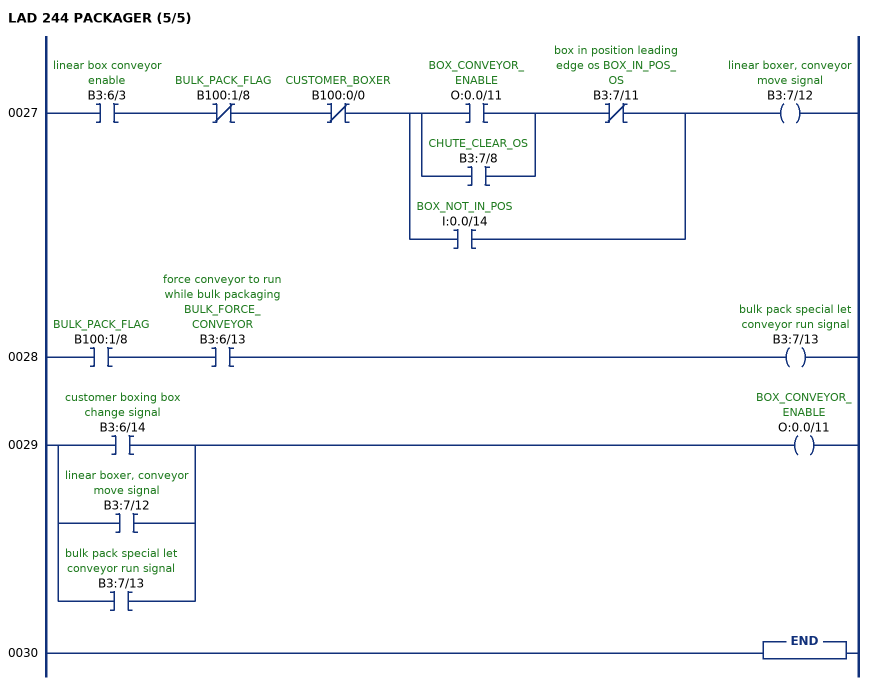
% Rung: 27 %
SOR XIC B3:6/3 XIO B100:1/8 XIO B100:0/0 BST BST XIC O:0.0/11 NXB XIC B3:7/8 BND XIO B3:7/11 NXB XIC I:0.0/14 BND OTE B3:7/12 EOR
%   B3:6/3  "linear box conveyor enable" %
%   B100:1/8  BULK_PACK_FLAG %
%   B100:0/0  CUSTOMER_BOXER %
%   O:0.0/11  BOX_CONVEYOR_ENABLE %
%   B3:7/8  CHUTE_CLEAR_OS %
%   B3:7/11  BOX_IN_POS_OS  "box in position leading edge os" %
%   I:0.0/14  BOX_NOT_IN_POS %
%   B3:7/12  "linear boxer, conveyor move signal" %
% Rung: 28 %
SOR XIC B100:1/8 XIC B3:6/13 OTE B3:7/13 EOR
%   B100:1/8  BULK_PACK_FLAG %
%   B3:6/13  BULK_FORCE_CONVEYOR  "force conveyor to run while bulk packaging" %
%   B3:7/13  "bulk pack special let conveyor run signal" %
% Rung: 29 %
SOR BST XIC B3:6/14 NXB XIC B3:7/12 NXB XIC B3:7/13 BND OTE O:0.0/11 EOR
%   B3:6/14  "customer boxing box change signal" %
%   B3:7/12  "linear boxer, conveyor move signal" %
%   B3:7/13  "bulk pack special let conveyor run signal" %
%   O:0.0/11  BOX_CONVEYOR_ENABLE %
% Rung: 30 %
SOR END EOR

LADDER 245 "NO PACKAGE"
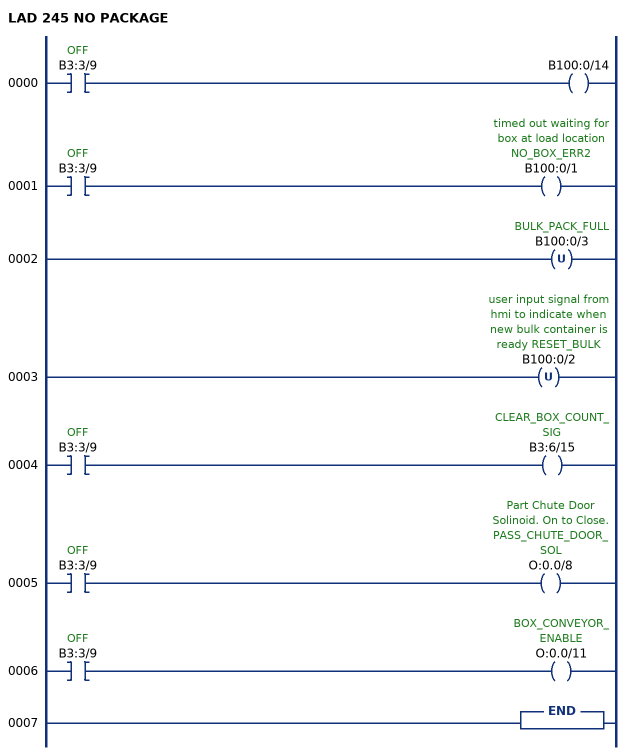
% Rung: 0 %
SOR XIC B3:3/9 OTE B100:0/14 EOR
%   B3:3/9  OFF %
% Rung: 1 %
SOR XIC B3:3/9 OTE B100:0/1 EOR
%   B3:3/9  OFF %
%   B100:0/1  NO_BOX_ERR2  "timed out waiting for box at load location" %
% Rung: 2 %
SOR OTU B100:0/3 EOR
%   B100:0/3  BULK_PACK_FULL %
% Rung: 3 %
SOR OTU B100:0/2 EOR
%   B100:0/2  RESET_BULK  "user input signal from hmi to indicate when new bulk container is ready" %
% Rung: 4 %
SOR XIC B3:3/9 OTE B3:6/15 EOR
%   B3:3/9  OFF %
%   B3:6/15  CLEAR_BOX_COUNT_SIG %
% Rung: 5 %
SOR XIC B3:3/9 OTE O:0.0/8 EOR
%   B3:3/9  OFF %
%   O:0.0/8  PASS_CHUTE_DOOR_SOL  "Part Chute Door Solinoid. On to Close." %
% Rung: 6 %
SOR XIC B3:3/9 OTE O:0.0/11 EOR
%   B3:3/9  OFF %
%   O:0.0/11  BOX_CONVEYOR_ENABLE %
% Rung: 7 %
SOR END EOR

LADDER 246 "RATE1"
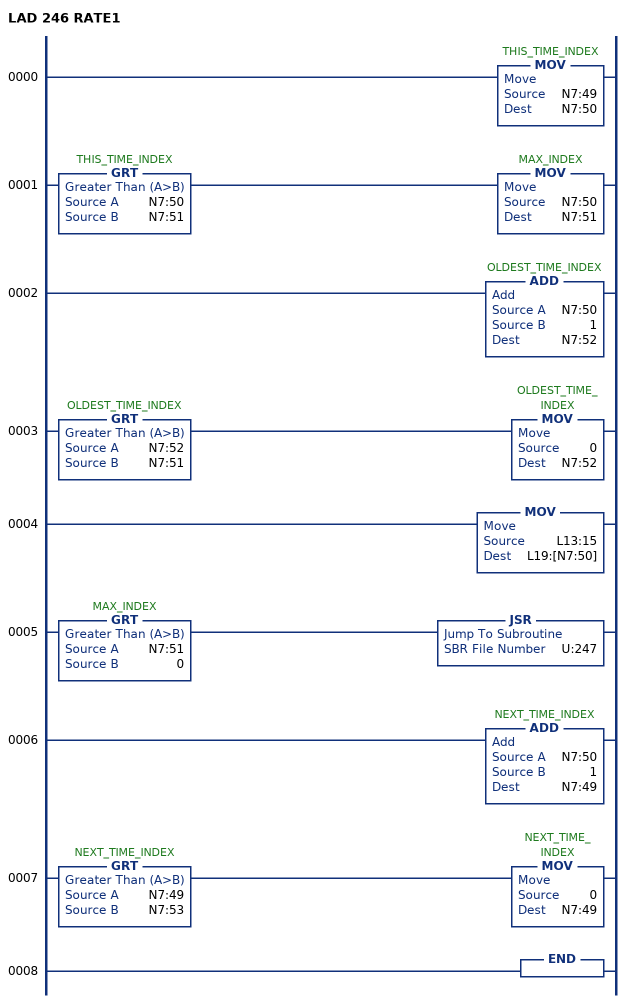
% Rung: 0 %
SOR MOV N7:49 N7:50 EOR
%   N7:49  NEXT_TIME_INDEX %
%   N7:50  THIS_TIME_INDEX %
% Rung: 1 %
SOR GRT N7:50 N7:51 MOV N7:50 N7:51 EOR
%   N7:50  THIS_TIME_INDEX %
%   N7:51  MAX_INDEX %
% Rung: 2 %
SOR ADD N7:50 1 N7:52 EOR
%   N7:50  THIS_TIME_INDEX %
%   N7:52  OLDEST_TIME_INDEX %
% Rung: 3 %
SOR GRT N7:52 N7:51 MOV 0 N7:52 EOR
%   N7:52  OLDEST_TIME_INDEX %
%   N7:51  MAX_INDEX %
% Rung: 4 %
SOR MOV L13:15 L19:[N7:50] EOR
%   L13:15  THE_TIME %
%   N7:50  THIS_TIME_INDEX %
% Rung: 5 %
SOR GRT N7:51 0 JSR U:247 EOR
%   N7:51  MAX_INDEX %
% Rung: 6 %
SOR ADD N7:50 1 N7:49 EOR
%   N7:50  THIS_TIME_INDEX %
%   N7:49  NEXT_TIME_INDEX %
% Rung: 7 %
SOR GRT N7:49 N7:53 MOV 0 N7:49 EOR
%   N7:49  NEXT_TIME_INDEX %
%   N7:53  UPPER_INDEX_LIMIT %
% Rung: 8 %
SOR END EOR

LADDER 247 "RATE2"
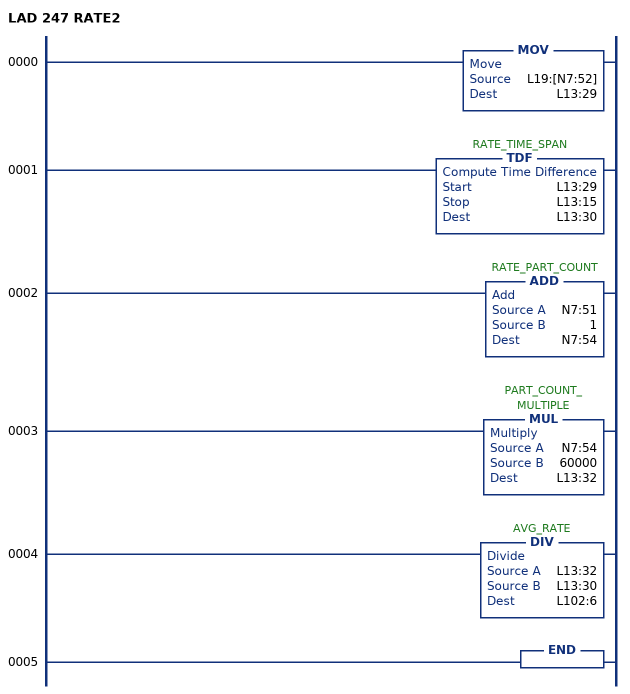
% Rung: 0 %
SOR MOV L19:[N7:52] L13:29 EOR
%   N7:52  OLDEST_TIME_INDEX %
% Rung: 1 %
SOR TDF L13:29 L13:15 L13:30 EOR
%   L13:15  THE_TIME %
%   L13:30  RATE_TIME_SPAN %
% Rung: 2 %
SOR ADD N7:51 1 N7:54 EOR
%   N7:51  MAX_INDEX %
%   N7:54  RATE_PART_COUNT %
% Rung: 3 %
SOR MUL N7:54 60000 L13:32 EOR
%   N7:54  RATE_PART_COUNT %
%   L13:32  PART_COUNT_MULTIPLE %
% Rung: 4 %
SOR DIV L13:32 L13:30 L102:6 EOR
%   L13:32  PART_COUNT_MULTIPLE %
%   L13:30  RATE_TIME_SPAN %
%   L102:6  AVG_RATE %
% Rung: 5 %
SOR END EOR

LADDER 248 "RESET RATE"
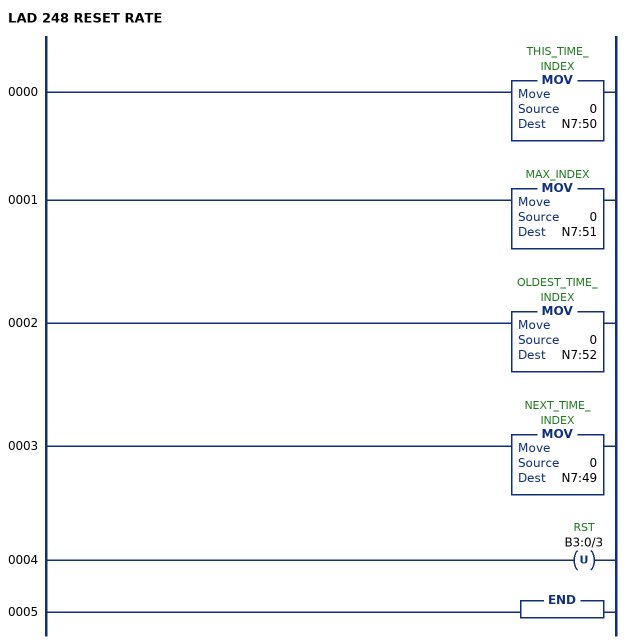
% Rung: 0 %
SOR MOV 0 N7:50 EOR
%   N7:50  THIS_TIME_INDEX %
% Rung: 1 %
SOR MOV 0 N7:51 EOR
%   N7:51  MAX_INDEX %
% Rung: 2 %
SOR MOV 0 N7:52 EOR
%   N7:52  OLDEST_TIME_INDEX %
% Rung: 3 %
SOR MOV 0 N7:49 EOR
%   N7:49  NEXT_TIME_INDEX %
% Rung: 4 %
SOR OTU B3:0/3 EOR
%   B3:0/3  RST %
% Rung: 5 %
SOR END EOR

LADDER 249 "NP STOP"    % stop on no good %
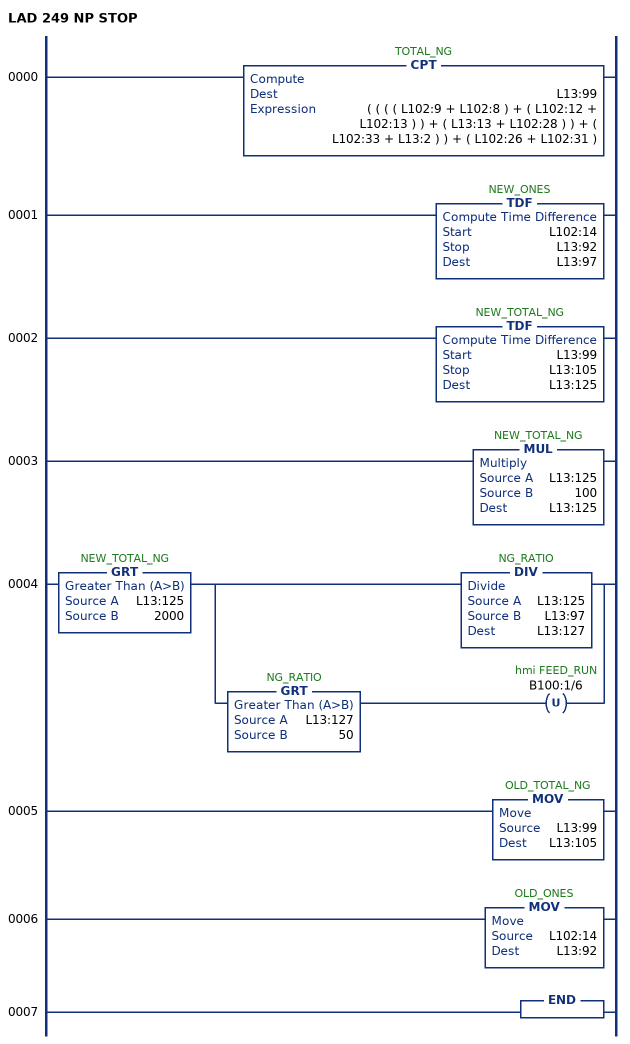
% Rung: 0 %
SOR CPT L13:99 " ( ( ( ( L102:9 + L102:8 ) + ( L102:12 + L102:13 ) ) + ( L13:13 + L102:28 ) ) + ( L102:33 + L13:2 ) ) + ( L102:26 + L102:31 ) " EOR
%   L13:99  TOTAL_NG %
%   L102:9  "too wide bottom" %
%   L102:8  "too close bottom" %
%   L102:12  "too close top count" %
%   L102:13  "too wide top count" %
%   L102:28  I1_I5_SKIPPEDCOUNT %
%   L102:33  I2_I6_SKIPPEDCOUNT %
%   L102:26  I1_I5_FAIL_COUNT %
%   L102:31  I2_I6_FAIL_COUNT %
% Rung: 1 %
SOR TDF L102:14 L13:92 L13:97 EOR
%   L102:14  ONES %
%   L13:92  OLD_ONES %
%   L13:97  NEW_ONES %
% Rung: 2 %
SOR TDF L13:99 L13:105 L13:125 EOR
%   L13:99  TOTAL_NG %
%   L13:105  OLD_TOTAL_NG %
%   L13:125  NEW_TOTAL_NG %
% Rung: 3 %
SOR MUL L13:125 100 L13:125 EOR
%   L13:125  NEW_TOTAL_NG %
% Rung: 4 %
SOR GRT L13:125 2000 BST DIV L13:125 L13:97 L13:127 NXB GRT L13:127 50 OTU B100:1/6 BND EOR
%   L13:125  NEW_TOTAL_NG %
%   L13:97  NEW_ONES %
%   L13:127  NG_RATIO %
%   B100:1/6  FEED_RUN  "hmi" %
% Rung: 5 %
SOR MOV L13:99 L13:105 EOR
%   L13:99  TOTAL_NG %
%   L13:105  OLD_TOTAL_NG %
% Rung: 6 %
SOR MOV L102:14 L13:92 EOR
%   L102:14  ONES %
%   L13:92  OLD_ONES %
% Rung: 7 %
SOR END EOR

LADDER 250 "SPEED BOT"    % high speed %
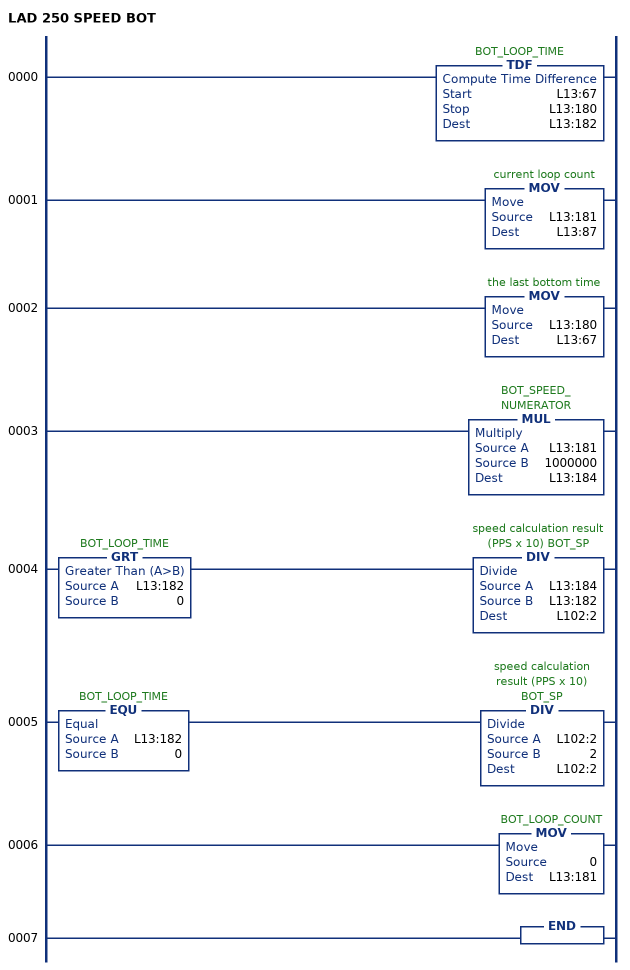
% Rung: 0 %
SOR TDF L13:67 L13:180 L13:182 EOR
%   L13:67  "the last bottom time" %
%   L13:180  BOT_THIS_TIME  "rtc bot belt movement event time" %
%   L13:182  BOT_LOOP_TIME %
% Rung: 1 %
SOR MOV L13:181 L13:87 EOR
%   L13:181  BOT_LOOP_COUNT %
%   L13:87  "current loop count" %
% Rung: 2 %
SOR MOV L13:180 L13:67 EOR
%   L13:180  BOT_THIS_TIME  "rtc bot belt movement event time" %
%   L13:67  "the last bottom time" %
% Rung: 3 %
SOR MUL L13:181 1000000 L13:184 EOR
%   L13:181  BOT_LOOP_COUNT %
%   L13:184  BOT_SPEED_NUMERATOR %
% Rung: 4 %
SOR GRT L13:182 0 DIV L13:184 L13:182 L102:2 EOR
%   L13:182  BOT_LOOP_TIME %
%   L13:184  BOT_SPEED_NUMERATOR %
%   L102:2  BOT_SP  "speed calculation result (PPS x 10)" %
% Rung: 5 %
SOR EQU L13:182 0 DIV L102:2 2 L102:2 EOR
%   L13:182  BOT_LOOP_TIME %
%   L102:2  BOT_SP  "speed calculation result (PPS x 10)" %
% Rung: 6 %
SOR MOV 0 L13:181 EOR
%   L13:181  BOT_LOOP_COUNT %
% Rung: 7 %
SOR END EOR

LADDER 251 "SPEED TOP"    % high speed %
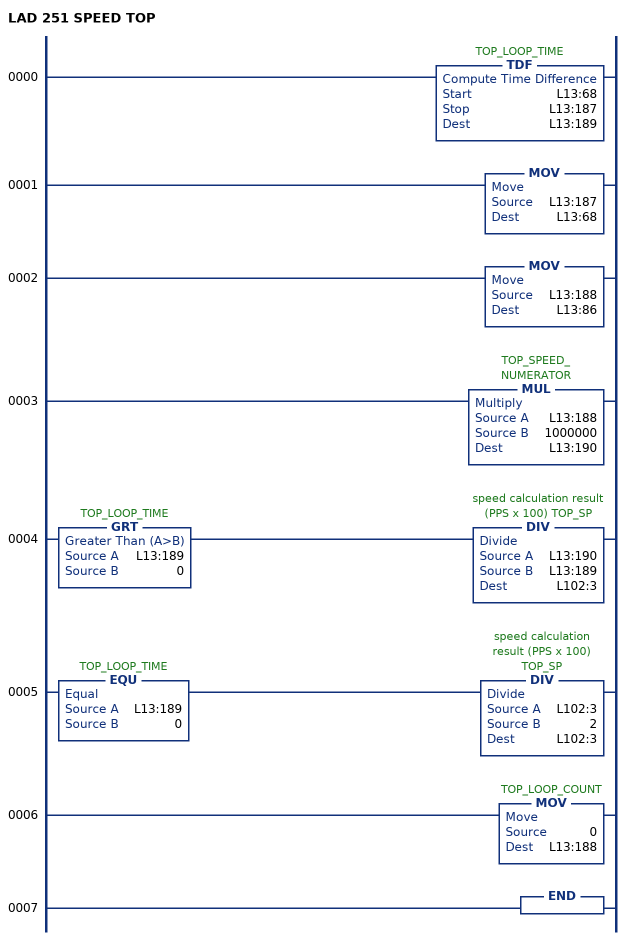
% Rung: 0 %
SOR TDF L13:68 L13:187 L13:189 EOR
%   L13:187  TOP_THIS_TIME  "rtc top belt movement event time" %
%   L13:189  TOP_LOOP_TIME %
% Rung: 1 %
SOR MOV L13:187 L13:68 EOR
%   L13:187  TOP_THIS_TIME  "rtc top belt movement event time" %
% Rung: 2 %
SOR MOV L13:188 L13:86 EOR
%   L13:188  TOP_LOOP_COUNT %
% Rung: 3 %
SOR MUL L13:188 1000000 L13:190 EOR
%   L13:188  TOP_LOOP_COUNT %
%   L13:190  TOP_SPEED_NUMERATOR %
% Rung: 4 %
SOR GRT L13:189 0 DIV L13:190 L13:189 L102:3 EOR
%   L13:189  TOP_LOOP_TIME %
%   L13:190  TOP_SPEED_NUMERATOR %
%   L102:3  TOP_SP  "speed calculation result (PPS x 100)" %
% Rung: 5 %
SOR EQU L13:189 0 DIV L102:3 2 L102:3 EOR
%   L13:189  TOP_LOOP_TIME %
%   L102:3  TOP_SP  "speed calculation result (PPS x 100)" %
% Rung: 6 %
SOR MOV 0 L13:188 EOR
%   L13:188  TOP_LOOP_COUNT %
% Rung: 7 %
SOR END EOR

LADDER 252 "P BOT"    % high speed %
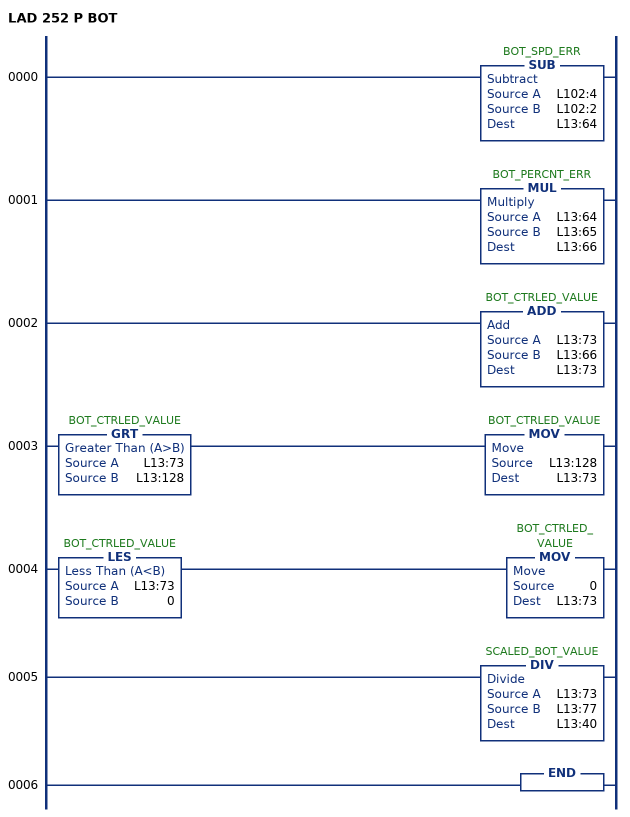
% Rung: 0 %
SOR SUB L102:4 L102:2 L13:64 EOR
%   L102:4  BOT_SPD_SETPOINT %
%   L102:2  BOT_SP  "speed calculation result (PPS x 10)" %
%   L13:64  BOT_SPD_ERR %
% Rung: 1 %
SOR MUL L13:64 L13:65 L13:66 EOR
%   L13:64  BOT_SPD_ERR %
%   L13:65  POS5SHIFT %
%   L13:66  BOT_PERCNT_ERR %
% Rung: 2 %
SOR ADD L13:73 L13:66 L13:73 EOR
%   L13:73  BOT_CTRLED_VALUE %
%   L13:66  BOT_PERCNT_ERR %
% Rung: 3 %
SOR GRT L13:73 L13:128 MOV L13:128 L13:73 EOR
%   L13:73  BOT_CTRLED_VALUE %
%   L13:128  "how much top has shifted since measurment" %
% Rung: 4 %
SOR LES L13:73 0 MOV 0 L13:73 EOR
%   L13:73  BOT_CTRLED_VALUE %
% Rung: 5 %
SOR DIV L13:73 L13:77 L13:40 EOR
%   L13:73  BOT_CTRLED_VALUE %
%   L13:40  SCALED_BOT_VALUE %
% Rung: 6 %
SOR END EOR

LADDER 253 "P TOP"    % high speed %
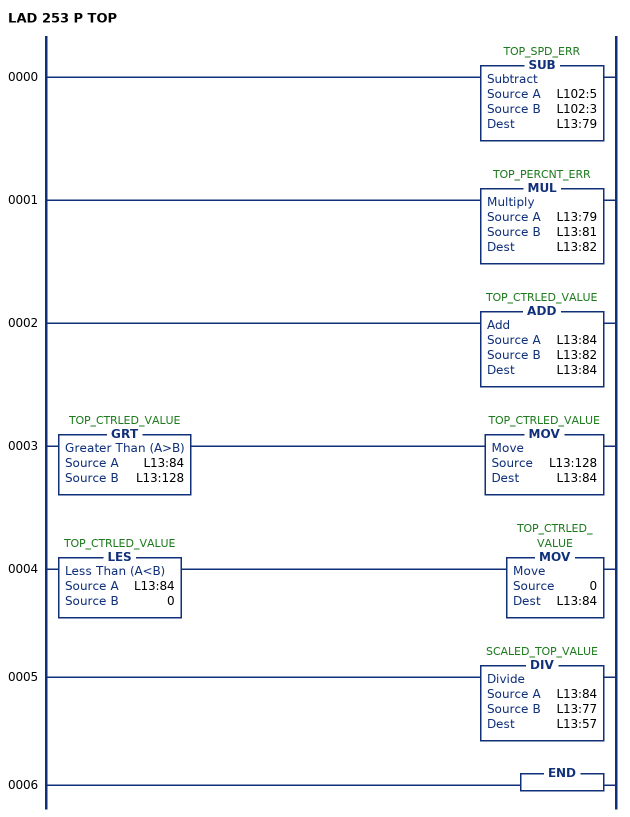
% Rung: 0 %
SOR SUB L102:5 L102:3 L13:79 EOR
%   L102:5  TOP_SPD_SETPOINT %
%   L102:3  TOP_SP  "speed calculation result (PPS x 100)" %
%   L13:79  TOP_SPD_ERR %
% Rung: 1 %
SOR MUL L13:79 L13:81 L13:82 EOR
%   L13:79  TOP_SPD_ERR %
%   L13:81  TOP_FDBK_RATIO %
%   L13:82  TOP_PERCNT_ERR %
% Rung: 2 %
SOR ADD L13:84 L13:82 L13:84 EOR
%   L13:84  TOP_CTRLED_VALUE %
%   L13:82  TOP_PERCNT_ERR %
% Rung: 3 %
SOR GRT L13:84 L13:128 MOV L13:128 L13:84 EOR
%   L13:84  TOP_CTRLED_VALUE %
%   L13:128  "how much top has shifted since measurment" %
% Rung: 4 %
SOR LES L13:84 0 MOV 0 L13:84 EOR
%   L13:84  TOP_CTRLED_VALUE %
% Rung: 5 %
SOR DIV L13:84 L13:77 L13:57 EOR
%   L13:84  TOP_CTRLED_VALUE %
%   L13:57  SCALED_TOP_VALUE %
% Rung: 6 %
SOR END EOR

LADDER 254 "TOTALCOUNT"
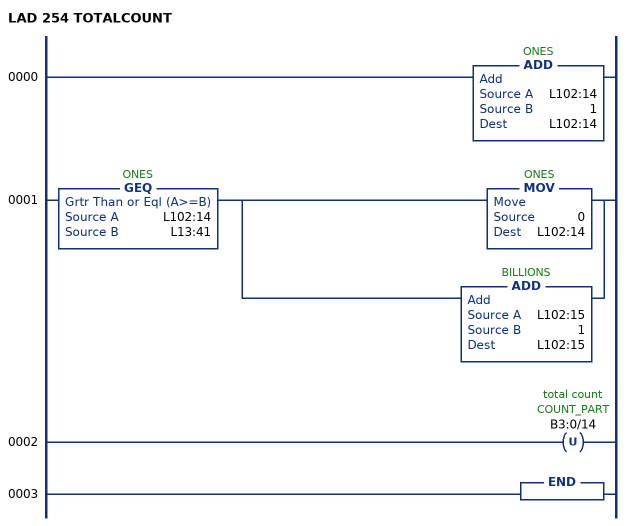
% Rung: 0 %
SOR ADD L102:14 1 L102:14 EOR
%   L102:14  ONES %
% Rung: 1 %
SOR GEQ L102:14 L13:41 BST MOV 0 L102:14 NXB ADD L102:15 1 L102:15 BND EOR
%   L102:14  ONES %
%   L13:41  "skipped count change in the last 3 seconds" %
%   L102:15  BILLIONS %
% Rung: 2 %
SOR OTU B3:0/14 EOR
%   B3:0/14  COUNT_PART  "total count" %
% Rung: 3 %
SOR END EOR

LADDER 255 "SAVED"
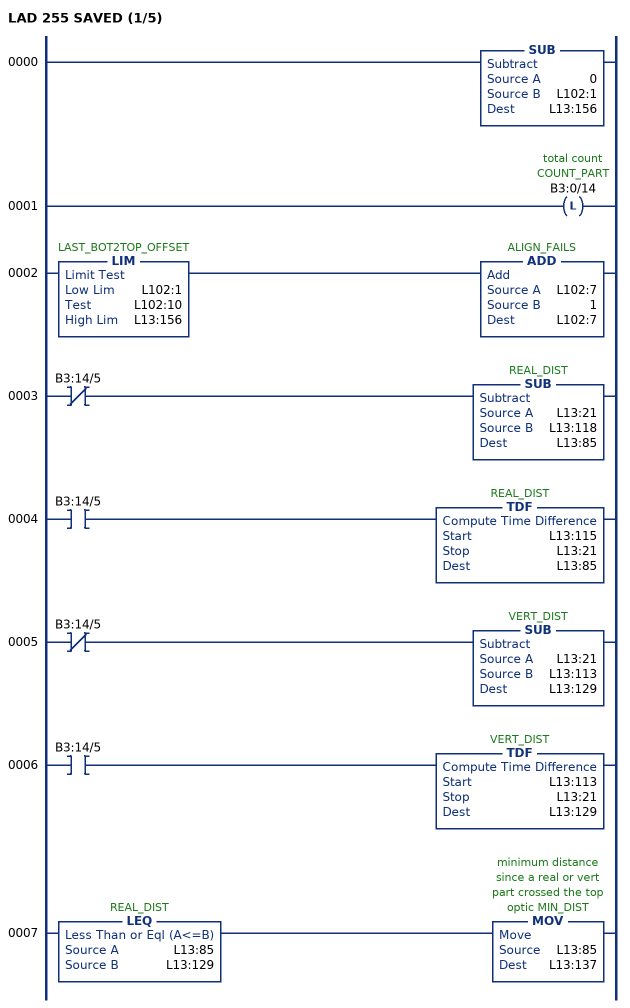
% Rung: 0 %
SOR SUB 0 L102:1 L13:156 EOR
%   L102:1  MAX_OFFSET  "transition zone width" %
% Rung: 1 %
SOR OTL B3:0/14 EOR
%   B3:0/14  COUNT_PART  "total count" %
% Rung: 2 %
SOR LIM L102:1 L102:10 L13:156 ADD L102:7 1 L102:7 EOR
%   L102:1  MAX_OFFSET  "transition zone width" %
%   L102:10  LAST_BOT2TOP_OFFSET %
%   L102:7  ALIGN_FAILS %
% Rung: 3 %
SOR XIO B3:14/5 SUB L13:21 L13:118 L13:85 EOR
%   L13:21  TOP_POSITION %
%   L13:118  REAL_CL_POSITION  "real part center line in raw position" %
%   L13:85  REAL_DIST %
% Rung: 4 %
SOR XIC B3:14/5 TDF L13:115 L13:21 L13:85 EOR
%   L13:115  TRAILING_EDGE_POS  "top optic trailing edge position" %
%   L13:21  TOP_POSITION %
%   L13:85  REAL_DIST %
% Rung: 5 %
SOR XIO B3:14/5 SUB L13:21 L13:113 L13:129 EOR
%   L13:21  TOP_POSITION %
%   L13:113  VIRT_CL_POSITION  "virtual part center line transfer from the bottom in raw position" %
%   L13:129  VERT_DIST %
% Rung: 6 %
SOR XIC B3:14/5 TDF L13:113 L13:21 L13:129 EOR
%   L13:113  VIRT_CL_POSITION  "virtual part center line transfer from the bottom in raw position" %
%   L13:21  TOP_POSITION %
%   L13:129  VERT_DIST %
% Rung: 7 %
SOR LEQ L13:85 L13:129 MOV L13:85 L13:137 EOR
%   L13:85  REAL_DIST %
%   L13:129  VERT_DIST %
%   L13:137  MIN_DIST  "minimum distance since a real or vert part crossed the top optic" %

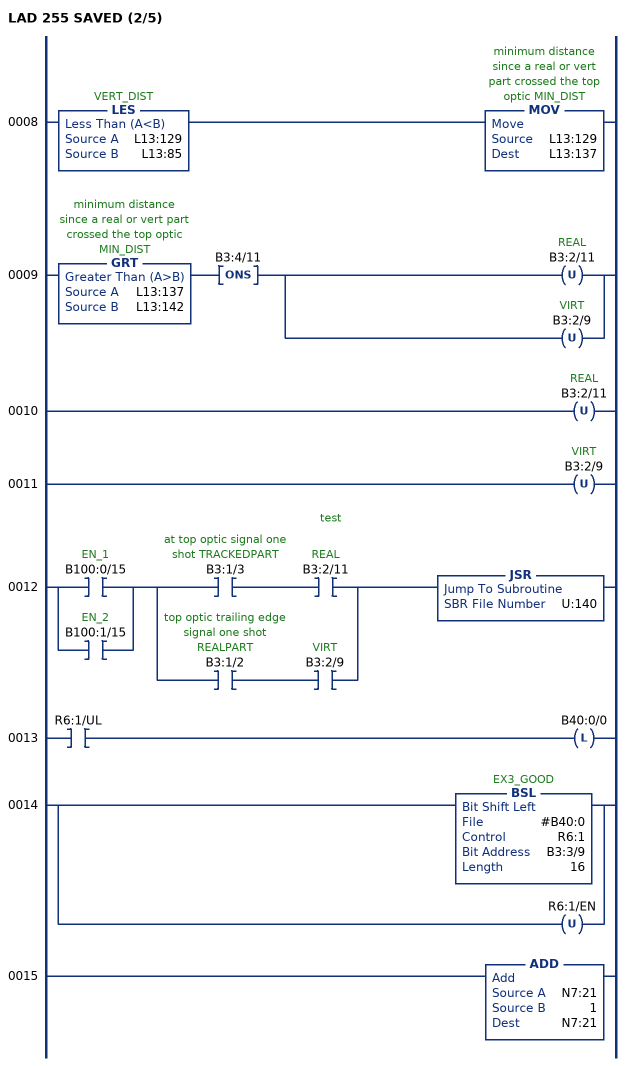
% Rung: 8 %
SOR LES L13:129 L13:85 MOV L13:129 L13:137 EOR
%   L13:129  VERT_DIST %
%   L13:85  REAL_DIST %
%   L13:137  MIN_DIST  "minimum distance since a real or vert part crossed the top optic" %
% Rung: 9 %
SOR GRT L13:137 L13:142 ONS B3:4/11 BST OTU B3:2/11 NXB OTU B3:2/9 BND EOR
%   L13:137  MIN_DIST  "minimum distance since a real or vert part crossed the top optic" %
%   L13:142  LAST_ALIGNMENT_FAILS %
%   B3:2/11  REAL %
%   B3:2/9  VIRT %
% Rung: 10 %
SOR OTU B3:2/11 EOR
%   B3:2/11  REAL %
% Rung: 11 %
SOR OTU B3:2/9 EOR
%   B3:2/9  VIRT %
% Rung: 12 %
% test %
SOR BST XIC B100:0/15 NXB XIC B100:1/15 BND BST XIC B3:1/3 XIC B3:2/11 NXB XIC B3:1/2 XIC B3:2/9 BND JSR U:140 EOR
%   B100:0/15  EN_1 %
%   B100:1/15  EN_2 %
%   B3:1/3  TRACKEDPART  "at top optic signal one shot" %
%   B3:2/11  REAL %
%   B3:1/2  REALPART  "top optic trailing edge signal one shot" %
%   B3:2/9  VIRT %
% Rung: 13 %
SOR XIC R6:1/UL OTL B40:0/0 EOR
% Rung: 14 %
SOR BST BSL #B40:0 R6:1 B3:3/9 16 NXB OTU R6:1/EN BND EOR
%   B40:0  EX3_GOOD %
%   B3:3/9  OFF %
% Rung: 15 %
SOR ADD N7:21 1 N7:21 EOR

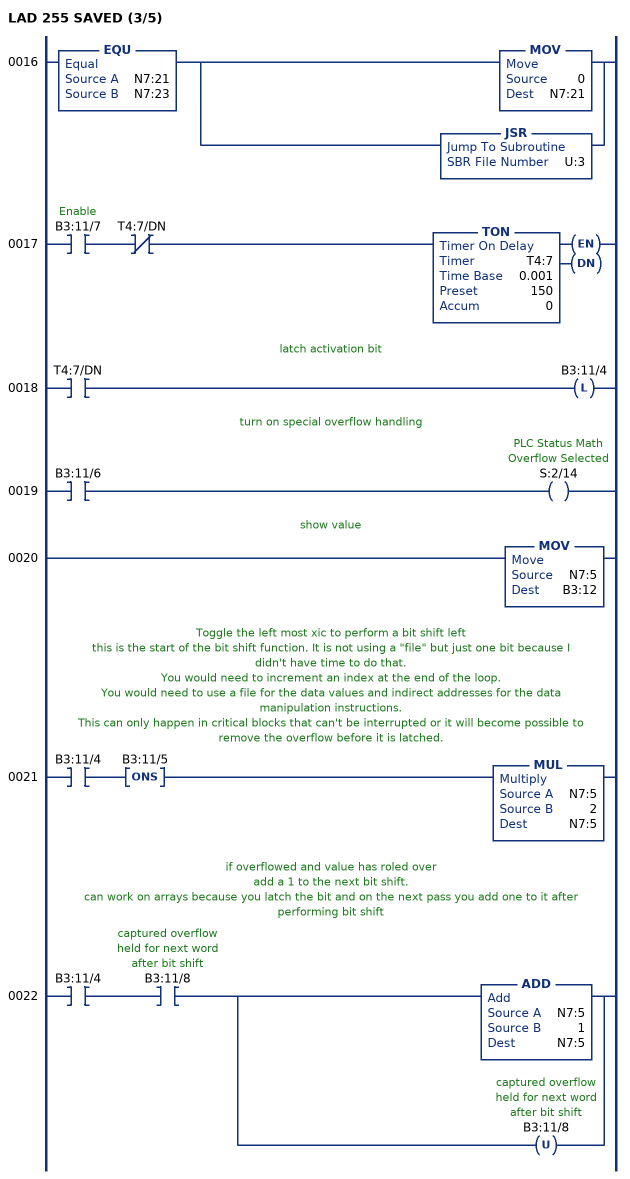
% Rung: 16 %
SOR EQU N7:21 N7:23 BST MOV 0 N7:21 NXB JSR U:3 BND EOR
% Rung: 17 %
SOR XIC B3:11/7 XIO T4:7/DN TON T4:7 0.001 150 0 EOR
%   B3:11/7  "Enable" %
% Rung: 18 %
% latch activation bit %
SOR XIC T4:7/DN OTL B3:11/4 EOR
% Rung: 19 %
% turn on special overflow handling %
SOR XIC B3:11/6 OTE S:2/14 EOR
%   S:2/14  "PLC Status Math Overflow Selected" %
% Rung: 20 %
% show value %
SOR MOV N7:5 B3:12 EOR
% Rung: 21 %
% Toggle the left most xic to perform a bit shift left
% 
% this is the start of the bit shift function. It is not using a "file" but just one bit because I didn't have time to do that.
% You would need to increment an index at the end of the loop.
% You would need to use a file for the data values and indirect addresses for the data manipulation instructions.
% 
% This can only happen in critical blocks that can't be interrupted or it will become possible to remove the overflow before it is latched. %
SOR XIC B3:11/4 ONS B3:11/5 MUL N7:5 2 N7:5 EOR
% Rung: 22 %
% if overflowed and value has roled over
% add a 1 to the next bit shift.
% can work on arrays because you latch the bit and on the next pass you add one to it after performing bit shift %
SOR XIC B3:11/4 XIC B3:11/8 BST ADD N7:5 1 N7:5 NXB OTU B3:11/8 BND EOR
%   B3:11/8  "captured overflow held for next word after bit shift" %

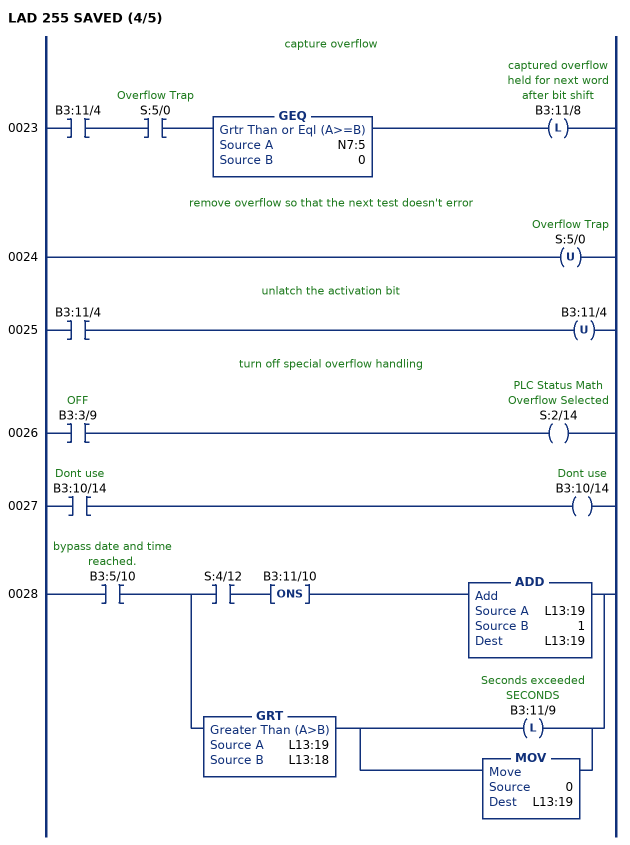
% Rung: 23 %
% capture overflow %
SOR XIC B3:11/4 XIC S:5/0 GEQ N7:5 0 OTL B3:11/8 EOR
%   S:5/0  "Overflow Trap" %
%   B3:11/8  "captured overflow held for next word after bit shift" %
% Rung: 24 %
% remove overflow so that the next test doesn't error %
SOR OTU S:5/0 EOR
%   S:5/0  "Overflow Trap" %
% Rung: 25 %
% unlatch the activation bit %
SOR XIC B3:11/4 OTU B3:11/4 EOR
% Rung: 26 %
% turn off special overflow handling %
SOR XIC B3:3/9 OTE S:2/14 EOR
%   B3:3/9  OFF %
%   S:2/14  "PLC Status Math Overflow Selected" %
% Rung: 27 %
SOR XIC B3:10/14 OTE B3:10/14 EOR
%   B3:10/14  "Dont use" %
% Rung: 28 %
SOR XIC B3:5/10 BST XIC S:4/12 ONS B3:11/10 ADD L13:19 1 L13:19 NXB GRT L13:19 L13:18 BST OTL B3:11/9 NXB MOV 0 L13:19 BND BND EOR
%   B3:5/10  "bypass date and time reached." %
%   L13:18  MAX %
%   B3:11/9  SECONDS  "Seconds exceeded" %

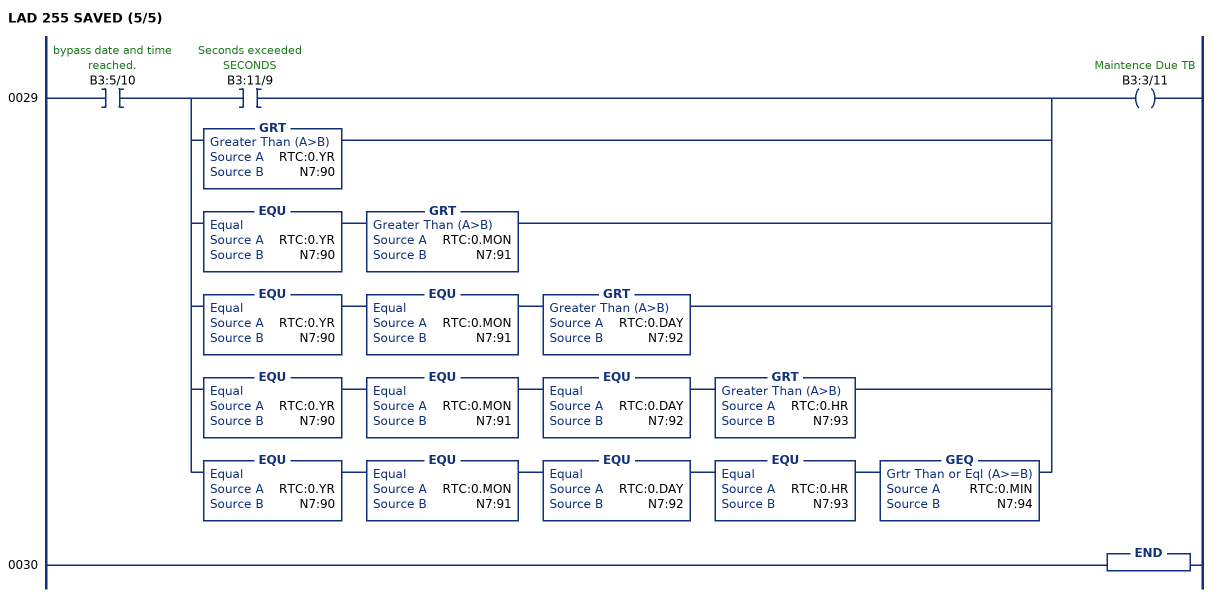
% Rung: 29 %
SOR XIC B3:5/10 BST XIC B3:11/9 NXB GRT RTC:0.YR N7:90 NXB EQU RTC:0.YR N7:90 GRT RTC:0.MON N7:91 NXB EQU RTC:0.YR N7:90 EQU RTC:0.MON N7:91 GRT RTC:0.DAY N7:92 NXB EQU RTC:0.YR N7:90 EQU RTC:0.MON N7:91 EQU RTC:0.DAY N7:92 GRT RTC:0.HR N7:93 NXB EQU RTC:0.YR N7:90 EQU RTC:0.MON N7:91 EQU RTC:0.DAY N7:92 EQU RTC:0.HR N7:93 GEQ RTC:0.MIN N7:94 BND OTE B3:3/11 EOR
%   B3:5/10  "bypass date and time reached." %
%   B3:11/9  SECONDS  "Seconds exceeded" %
%   N7:90  RTC %
%   B3:3/11  TB  "Maintence Due" %
% Rung: 30 %
SOR END EOR

OTHER DOCUMENTED ADDRESSES
  B38:0  EX1_GOOD
  B189:0/0  "change box"
  B189:0/9  "override boxing ok or not full signal"
  B189:0/11  "HMI force door close"
  B196:1/0  "Chute door is closed"
  B196:1/1  "control chute door"
  B196:1/13  "force box conveyor on"
  B196:3/0  "for hmi to continue production unlatched by hmi"
  HSC:0.0  "top"
  HSC:0.3/6  "Underflow interrupt"
  HSC:0.3/7  "Overflow interrupt"
  HSC:1.0  "bot"
  HSC:1.3/6  "Underflow interrupt"
  HSC:1.3/7  "Overflow interrupt"
  I7_TRAC  
  I:0.0/0  TOP_EN  "Encoder Signal Top"
  I:0.0/4  BOT_EN  "Encoder Signal Bot"
  I:0.1/4  "not used"
  I:0.1/5  "not used"
  I:0.1/6  "not used"
  I:0.1/7  "not used"
  I:0.1/8  "not used"
  I:0.1/9  "not used"
  I:0.1/10  "not used"
  I:0.1/11  "not used"
  I:0.1/12  "not used"
  I:0.1/13  "not used"
  I:0.1/14  "not used"
  I:0.1/15  "not used"
  I:0.2  "not used"
  I:0.3  "not used"
  I:0.4  "Spare Analog Input 1"
  I:0.5  "Spare Analog Input 2"
  I:0.6  "Spare Analog Input 3"
  I:2.0/0  FRONT_ESTOP
  I:2.0/1  REAR_ESTOP
  I:2.0/3  BOX_CNV_NOT_FULL  "input turns off when box discharge full optics are blocked"
  I:2.0/4  "this input is on when a box is not in position"
  I:2.0/8  FRONT_DOOR  "front door signal ce models only"
  I:2.0/9  REAR_DOOR  "rear door signal ce models only"
  I:2.0/11  "spare"
  L13:132  "set speed"
  L13:133  "controlled speed"
  L13:183  TKS_PER_SECOND
  L23:19  TOP_OPT_FAIL_CT
  L23:34  AIR_PRESSURE_FAULT
  L28:0  INS_1_TIME
  L29:0  INS_1_POS
  L30:0  INS_5_TIME
  L31:0  INS_5_POS
  L32:0  INS_6_TIME
  L33:0  INS_6_POS
  L192:1  BOT_LAST_TIME  "rtc bot belt previous movement event time"
  L192:2  BOT_CYCLE_TIME  "rtc bot belt time between events"
  L192:7  FROM_REAL  "distance from real part signal at optic location"
  L192:8  FROM_TRACKED  "distance from tracked part signal at optic location"
  L192:16  TOP_LAST_TIME  "rtc top belt previous movement event time"
  L192:17  TOP_CYCLE_TIME  "rtc top belt time between events"
  L199:5  ACQTM51
  L199:6  ACQTM52
  L199:7  ACQTM53
  L199:9  "ones"
  L199:10  "billions"
  L199:13  DUMP_LONG
  L199:15  ACQTM11
  L199:16  ACQTM12
  L199:17  ACQTM13
  L199:20  RESULTTM1
  L199:22  CLEARTIME5COUNT
  L199:23  CLEARTIME6COUNT
  L199:24  ACQTM61
  L199:25  ACQTM62
  L199:26  ACQTM63
  L199:27  TMSINCETRIG1
  L199:29  TMSINCETRIG5
  L199:30  TMSINCETRIG6
  L199:31  CLEARTIME1COUNT
  L199:32  RESULTTM5
  L199:33  RESULTTM6
  L199:34  MAXACQTM1
  L199:36  MAXACQTM6
  N7  
  N101:2  I3_TRIG_LOC
  N101:3  I4_TRIG_LOC
  O:0.0/1  "spare"
  O:0.0/12  "not used"
  O:0.0/13  "not used"
  O:0.0/14  "not used"
  O:0.0/15  "not used"
  O:0.1  "not used"
  O:0.2  "not used"
  O:0.3  "not used"
  O:1.2  "Feeder Bowl Speed"
  O:3.0/1  "Part Chute Door Solinoid. On to Close."
  O:3.0/2  "spare"
  O:3.0/3  "light curtain range selection /* needed? */"
  O:3.0/7  "door unlocks on CE models"
  O:3.0/8  "Light?"
  O:3.0/9  NUT_HOPPER  "Nut Hopper Enable"
  O:3.0/11  NUT_FEEDER_AIR  "Nut Feeder Bowl Air Enable"
  O:3.0/12  BOLT_FEEDER  "feeder bowl output on = enable"
  PFILE:6  "check for part jams"
  PFILE:10  "Bottom belt HSC"
  PFILE:12  "Top belt HSC"
  Q2:55  END_OF_MAIN
  Q5:94  END_OF_BELTS
  T20:0  "Trigger On Time"
  U:9  "slow data"
  U:24  "check skipped fail rate"
  U:28  "faults"
  U:29  "speed"
  U:30  "count"
  U:31  "rate calc"
  U:32  "boxer"
  U:33  "bulk pack"
  U:34  "customer boxing unit signals"
  U:35  "cleanup"

COMMENTS NOT ATTACHED TO A CURRENT RUNG
  R6:2: B41 is the top good 3 file
  R6:6/DN: B35 is the top NG file
  R6:10/DN: B37 is the top good 1 file
  R6:11/DN: B39 is the top good 2 file
  B100:1/15: what is this code for?
  R6:0: B36 is the bottom GOOD file
  R6:10: B37 is the top good 1 file
  R6:6: B35 is the top NG file
  R6:4: B34 is the bottom NG file

REVISION NOTES
  13: updated count reset
  14: added io moduals
  15: multiple steps toward new hmi integration
  21: test
  27: fix error if bulk pack and no boxing fallout were on

DATA TABLE (non-zero values as saved)
DATA B3
% B3:0 % 0X8862 0X1141 0X4041 0X6101 0XECB7 0X1504 0X0438 0X0461 0X3FA0 0X2330
% B3:10 % 0X21F0 0X40C6 0X4000 0X10B4 0X4801 0X0000 0X0000 0X0000 0X0000 0X0000
% B3:50 % 0X0001 0X0000 0X0000 0X0000 0X0000 0X0000 0X0000 0X0000 0X0000 0X0000
DATA T4
% .PRE .ACC %
% T4:0 % 0 1
% T4:1 % 150 0
% T4:2 % 400 0
% T4:3 % 250 68
% T4:4 % 1000 1000
% T4:5 % 5 5
% T4:6 % 10 32766
% T4:7 % 150 0
% T4:8 % 20 0
% T4:9 % 50 34
% T4:10 % 200 200
% T4:11 % 111 0
% T4:12 % 30 30
% T4:13 % 250 0
% T4:14 % 666 0
% T4:15 % 1000 1002
% T4:16 % 400 0
% T4:17 % 100 11
% T4:18 % 5 0
% T4:19 % 300 0
% T4:20 % 200 0
% T4:21 % 200 0
% T4:22 % 200 0
% T4:23 % 250 0
% T4:24 % 666 0
% T4:25 % 666 0
% T4:26 % 666 0
% T4:27 % 250 0
% T4:28 % 250 0
% T4:29 % 5000 0
% T4:30 % 333 0
% T4:31 % 333 70
% T4:32 % 250 60
% T4:33 % 250 62
% T4:34 % 1111 0
% T4:35 % 23 0
DATA C5
% .PRE .ACC %
% C5:0 % 32766 0
DATA R6
% .LEN .POS %
% R6:0 % 1250 0
% R6:1 % 16 0
% R6:2 % 1050 0
% R6:3 % 1050 0
% R6:4 % 1250 0
% R6:5 % 1250 0
% R6:6 % 1713 0
% R6:7 % 16 0
% R6:8 % 1024 0
% R6:9 % 3 0
% R6:10 % 1713 0
% R6:11 % 1050 0
% R6:12 % 10 0
% R6:13 % 10 0
% R6:14 % 10 0
% R6:15 % 10 0
% R6:16 % 1713 0
% R6:17 % 1713 0
% R6:18 % 1050 0
% R6:19 % 10 0
DATA N7
% N7:0 % -20284 4 994 191 3 0 0 0 500 43
% N7:10 % 1000 43 0 8 22 22 1000 2000 50 1050
% N7:20 % 0 1329 16 2000 0 48 0 0 0 250
% N7:30 % 666 -17477 150 0 3071 1333 83 45 0 45
% N7:40 % 2 38 1 37 141 1266 32767 1266 0 16
% N7:50 % 15 16 16 16 17 813 100 0 0 3
% N7:60 % 1713 1713 1050 868 0 0 4999 5 400 400
% N7:70 % 100 200 300 400 90 190 290 390 -5467 20234
% N7:80 % 0 0 1348 1357 1398 1408 87 6 0 0
% N7:90 % 2011 4 4 12 1 87 6 222 222 12
% N7:100 % 1003 90 110 100 175 25 0 0 0 0
% N7:190 % -128 27477 27605 32767 0 0 0 0 0 0
DATA F8
% F8:0 % 6
DATA L13
% L13:0 % 245711 434202 0 245797 646432
% L13:5 % 44 188275 2256 648763 6
% L13:10 % 5 979645 0 15 90
% L13:15 % -312026727 -2147483648 2147483647 2147483647 82058
% L13:20 % 657699988 -893661244 777 -1022733994 100
% L13:25 % 0 -1023197984 0 0 -314845574
% L13:30 % 2818499 -1022733998 1020000 -316701426 1444
% L13:35 % 1 0 0 -1287730312 -1287730267
% L13:40 % 1778 1000000000 1000000 -316701472 -313711130
% L13:45 % -313711101 45 0 46 657699236
% L13:50 % 1684425 2256 -1542513552 0 0
% L13:55 % 1684396 195464051 1837 82392473 82399453
% L13:60 % 26975 1992914 0 600 11
% L13:65 % 8 88 -1287741880 -1287741882 2
% L13:70 % 579072579 584 8 177776 657699236
% L13:75 % 16 30 100 -1542514318 1
% L13:80 % 557730 6 6 40 183700
% L13:85 % 274296 168 168 0 1684465
% L13:90 % 1684436 3 284784 5 -313711085
% L13:95 % 99 14840 0 -313711056 15
% L13:100 % 100 7 -695148792 1111 450
% L13:105 % 15 568360 657699115 17674 657699108
% L13:110 % 7 33 66 -895201556 -894221915
% L13:115 % -894221907 8 4 -894221911 1000
% L13:120 % 43771938 9476 99 0 179
% L13:125 % 0 579072579 20400 409600 274297
% L13:130 % 33 66 0 249 -249
% L13:135 % 0 500 274296 1000 0
% L13:140 % 49 -49 36 50 50
% L13:145 % 2257 5 195464154 5 16
% L13:150 % 12 20 36290 -36290 979645
% L13:155 % 100 -10 0 48 4589052
% L13:160 % 15 45 45 1220 45
% L13:165 % -894221569 -894221559 -894221569 -894221559 6707
% L13:170 % 12817 28487 28486 300 300
% L13:175 % 4 4 524330 536870935 38
% L13:180 % -1287714512 90 51072 1000000 168000000
% L13:185 % 0 0 -1287714637 90 50927
% L13:190 % 168000000 67108864 0 0 0
% L13:195 % 0 0 0 0 134217728
% L13:200 % 33554432 0 0 18432 0
% L13:205 % 0 0 0 975215 2390474
% L13:220 % 0 0 512 0 0
% L13:225 % 0 1048576 0 0 0
% L13:230 % 4096 0 0 1024 0
% L13:235 % 0 2097152 512 0 0
% L13:245 % 0 0 0 561152 0
DATA L19
% L19:0 % -314838571 -314831446 -314824515 -314817287 -314809973
% L19:5 % -314802647 -314795183 -314788039 -314659270 -314647641
% L19:10 % -313920605 -313905388 -313894582 -313871370 -313740630
% L19:15 % -313712145 -314845574 0 0 0
% L19:20 % 0 0 0 0 88080384
% L19:25 % 0 1207959552 1 -1073741816 33587204
% L19:30 % 131072 0 -2147483648 0 -2147483648
% L19:40 % 0 0 0 0 1
% L19:45 % 256 0 0 0 5250
DATA L20
% L20:0 % -316595342 -316595088 -316594835 -316594581 -316594328
% L20:5 % -316594075 -316593822 -316593569 -316593315 -316593060
% L20:10 % -316592806 -316592553 -316592299 -316592045 -316591791
% L20:15 % -316591536 -316591283 -316591029 -316590776 -316590523
% L20:20 % -316590133 -316590016 -316589761 -316589508 -316589254
% L20:25 % -316589000 -316588747 -316588493 -316576391 -315314954
% L20:30 % -315307247 -315300320 -315293494 -315286618 -315279323
% L20:35 % -315271918 -315264885 -315258036 -315250704 -315060108
% L20:40 % -315059855 -315059602 -315059348 -315059094 -315058840
% L20:45 % -315058586 -315058331 -315058076 -315030790 -314984369
% L20:50 % -314932686 -314924118 -314916890 -314909781 -314902170
% L20:55 % -314894705 -314887484 -314873694 -314866548 -314859624
% L20:60 % -314852408 -314844559 -314837555 -314830431 -314823500
% L20:65 % -314816271 -314808959 -314801632 -314794168 -314787023
% L20:70 % -314681008 -314658255 -314646626 -313919591 -313904373
% L20:75 % -313893567 -313870353 -313807301 -313807044 -313806789
% L20:80 % -313806534 -313806280 -313806024 -313805769 -313805516
% L20:85 % -313805262 -313739617 -313711130 -316598384 -316598132
% L20:90 % -316597878 -316597625 -316597372 -316597117 -316596864
% L20:95 % -316596611 -316596358 -316596104 -316595849 -316595595
% L20:100 % 200 524288 22 -2147483646 34
% L20:105 % 536870912 9 310378496 0 -1811939328
% L20:120 % 0 0 128 1073741824 0
% L20:125 % 0 0 0 1048576 0
% L20:130 % 1073741824 0 0 0 0
% L20:135 % 0 2048 0 0 0
% L20:145 % 0 0 0 0 268435456
% L20:150 % 0 512 0 0 0
% L20:165 % 0 0 1 0 131072
% L20:175 % 0 0 0 0 1048576
% L20:185 % 4194304 0 67108864 0 0
% L20:190 % 0 -2147483648 0 0 0
% L20:195 % 0 0 512 0 268435712
% L20:200 % 0 0 32768 0 0
% L20:210 % 8388608 0 0 0 0
% L20:225 % 16777216 0 0 4194304 0
% L20:235 % 64 68 0 128 16
% L20:240 % 0 0 0 64 0
% L20:250 % 0 0 0 671088640 1
% L20:255 % 171966464
DATA L21
% L21:0 % -895177776 -893998128 -895177776 -895177776 -895177776
% L21:5 % -559633456 -895177774 -626742320 -895177774 -291198000
% L21:10 % -895177774 -895177776 -895177766 -895177776 -895177774
% L21:15 % -895177776 -895173680 -895177776 -895095856 -895177776
% L21:20 % -895177772 -895177776 -895177740 -895177776 -895177736
% L21:25 % -895177776 -895177744 -895177776 -895158334 -894755098
% L21:30 % -894752534 -894750230 -894747959 -894745672 -894743246
% L21:35 % -894740783 -894738443 -894736165 -894733726 -894670324
% L21:40 % -894670240 -894670156 -894670071 -894669987 -894669902
% L21:45 % -894669817 -894669733 -894669648 -894660571 -894645129
% L21:50 % -894627936 -894625086 -894622682 -894620317 -894617785
% L21:55 % -894615302 -894612900 -894608313 -894605936 -894603632
% L21:60 % -894601231 -894598620 -894596290 -894593921 -894591615
% L21:65 % -894589210 -894586777 -894584340 -894581857 -894579480
% L21:70 % -894544211 -894536642 -894532774 -894290916 -894285854
% L21:75 % -894282259 -894274537 -894253562 -894253476 -894253392
% L21:80 % -894253307 -894253223 -894253137 -894253053 -894252968
% L21:85 % -894252884 -894231045 -894221569 -895177776 -895177776
% L21:90 % -895177776 -895177776 -895177776 -895177776 -895177776
% L21:95 % -895177776 -895177776 -895177776 -895177776 -895177776
% L21:110 % 0 4096 0 0 -2147483648
% L21:115 % 0 0 0 2048 0
% L21:120 % 0 0 262144 0 0
% L21:130 % 0 0 0 8388608 0
% L21:135 % 0 0 0 0 32
% L21:140 % 33554432 0 0 1024 0
% L21:145 % 0 0 0 0 1040
% L21:150 % 0 0 0 0 1073741824
% L21:155 % 0 0 0 0 524288
% L21:165 % 0 0 0 16384 32
% L21:170 % 8192 0 0 0 0
% L21:180 % 0 0 0 0 148
% L21:205 % 0 2048 0 0 0
% L21:210 % 0 0 0 75776 0
% L21:240 % 16 0 0 0 4
% L21:250 % 1024 0 0 0 32
DATA L22
% L22:0 % -313806255 -313806000 -313805745 -313805491 -313805237
% L22:5 % -313739587 -313711101 -315250674 -315060078 -315059823
% L22:10 % -315059567 -315059313 -315059059 -315058806 -315058551
% L22:15 % -315058298 -315058044 -315030760 -314984339 -314932656
% L22:20 % -314924088 -314916860 -314909751 -314902140 -314894675
% L22:25 % -314887454 -314873664 -314866518 -314859594 -314852378
% L22:30 % -314844529 -314837525 -314830401 -314823470 -314816241
% L22:35 % -314808928 -314801602 -314794138 -314786993 -314680978
% L22:40 % -314658225 -314646596 -313919561 -313904343 -313893537
% L22:45 % -313870323 -313807272 -313807018 -313806764 -313806509
DATA L23
% L23:0 % -894253214 -894253129 -894253045 -894252960 -894252876
% L23:5 % -894231035 -894221559 -894733716 -894670314 -894670229
% L23:10 % -894670144 -894670059 -894669975 -894669891 -894669806
% L23:15 % -894669722 -894669637 -894660561 -894645119 -894627926
% L23:20 % -894625076 -894622672 -894620307 -894617775 -894615292
% L23:25 % -894612890 -894608303 -894605926 -894603622 -894601221
% L23:30 % -894598610 -894596280 -894593911 -894591605 -894589200
% L23:35 % -894586767 -894584330 -894581847 -894579470 -894544201
% L23:40 % -894536632 -894532764 -894290906 -894285844 -894282249
% L23:45 % -894274527 -894253552 -894253468 -894253384 -894253299
DATA L30
% L30:0 % -316727498 -316727244 -316726989 -316726735 -316726480
% L30:5 % -316726226 -316725972 -316725718 -316725465 -316725212
% L30:10 % -316724957 -316724702 -316724447 -316724194 -316723939
% L30:15 % -316723685 -316723431 -316723177 -316722923 -316722667
% L30:20 % -316722414 -316722161 -316721906 -316721653 -316721400
% L30:25 % -316721146 -316720891 -316720636 -316720382 -316720127
% L30:30 % -316719873 -316719618 -316719364 -316719109 -316718854
% L30:35 % -316718600 -316718346 -316718093 -316717838 -316717583
% L30:40 % -316717328 -316717074 -316716821 -316716565 -316716312
% L30:45 % -316701472 -316728514 -316728260 -316728007 -316727752
DATA L31
% L31:0 % 657696600 657696600 657696600 657696600 657696600
% L31:5 % 657696600 657696600 657696600 657696600 657696600
% L31:10 % 657696600 657696600 657696600 657696600 657696600
% L31:15 % 657696600 657696600 657696600 657696600 657696600
% L31:20 % 657696600 657696600 657696600 657696600 657696600
% L31:25 % 657696600 657696600 657696600 657696600 657696600
% L31:30 % 657696600 657696600 657696600 657696600 657696600
% L31:35 % 657696600 657696600 657696600 657696600 657696600
% L31:40 % 657696600 657696600 657696600 657696600 657696600
% L31:45 % 657699236 657696600 657696600 657696600 657696600
DATA L32
% L32:0 % -1542513552 -1542513102 -1542514004 -1557910109 -1557909896
% L32:5 % -1557909688 -1557909474 -1557909271 -1557384768 -1557908847
% L32:10 % -1557908633 -1557908424 -1557908211 -1557907997 -1557907785
% L32:15 % -1557907586 -1557907374 -1557907159 -1557906946 -1557906759
% L32:20 % -1557906550 -1557906338 -1557906134 -1557905911 -1557905708
% L32:25 % -1557905494 -1557905285 -1557905066 -1557904859 -1557904640
% L32:30 % -1557904432 -1557904209 -1557903991 -1557903783 -1557903579
% L32:35 % -1557903367 -1557903159 -1557902951 -1557902743 -1557902539
% L32:40 % -1557902347 -1542622975 -1542622525 -1557912231 -1557912018
% L32:45 % -1557911805 -1557911591 -1557911383 -1557911170 -1557910951
DATA L33
% L33:0 % 847508784 579073578 579073077 575939187 575939230
% L33:5 % 575939272 575939315 575939356 575939399 575939441
% L33:10 % 575939484 575939526 575939569 575939612 575939655
% L33:15 % 575939695 575939738 575939781 575939824 575939862
% L33:20 % 575939904 575939947 575939988 575940033 575940074
% L33:25 % 575940117 575940159 575940203 575940245 575940289
% L33:30 % 575940331 575940376 575940420 575940462 575940503
% L33:35 % 575940546 575940588 575940630 575940672 575940713
% L33:40 % 575940752 579017052 579017281 575938759 575938802
% L33:45 % 575938845 575938888 575938930 575938973 -1571544631
DATA B34
% B34:0 % 0X0000 0X0000 0X0000 0X0000 0X8000 0X0000 0X0000 0X0000 0X0000 0X0000
% B34:40 % 0X0000 0X0000 0X0020 0X0000 0X0000 0X0000 0X0000 0X0000 0X0000 0X0000
% B34:60 % 0X0000 0X0000 0X0000 0X0000 0X0000 0X0000 0X0002 0X0000 0X0000 0X0000
% B34:110 % 0X0000 0X0000 0X0000 0X0000 0X0000 0X0000 0X0200 0X0000 0X0000 0X0000
% B34:120 % 0X0000 0X0000 0X0000 0X0000 0X0000 0X0000 0X0000 0X8000
DATA B35
% B35:110 % 0X0000 0X0000 0X0200 0X0000 0X0000 0X0000 0X0000 0X0000 0X0000 0X0000
DATA B36
% B36:50 % 0X0000 0X0000 0X0000 0X0000 0X2000 0X0000 0X0000 0X0000 0X0000 0X0000
DATA B37
% B37:0 % 0X0000 0X0000 0X2000 0X0000 0X0000 0X0000 0X0000 0X0000 0X0000 0X0000
DATA B40
% B40:0 % 0XAAAA
DATA B41
% B41:60 % 0X0000 0X0000 0X00AC 0X0000 0X0000 0X0000 0X0000 0X0000 0X0000 0X0000
DATA B100
% B100:0 % 0X2700 0X18A0 0X0004 0X0000 0X0000 0X0000 0X0000 0X0000 0X0000 0X0000
DATA N101
% N101:0 % 125 647 0 0 1178 100 990 1200 1200 1332
% N101:10 % 1342 1640 10 30144 3071 21297 1578 250 333 333
% N101:20 % 1000 500 400 0 0 0 250 250 0 0
DATA L102
% L102:0 % 30 10 3301 3297 3300
% L102:5 % 3300 0 0 0 0
% L102:10 % 0 5 0 0 284784
% L102:15 % 0 30 15 30 15
% L102:20 % 0 3 12 0 45
% L102:25 % 46 0 1 0 0
% L102:30 % 584 0 78947858 0 -1544775
% L102:35 % 0 500 0 999999 45
% L102:40 % 0 3 12 0 0
